// TIA Portal project "PROCESS OUTPUT" (V19)

(* hardware
DEVICE "SIMATIC 1200 station_1"  S71200.Device
   slot 0: "S7-1200 rack"  Rack  V1.0
   slot 1: "PLC_1"  CPU 1214C DC/DC/DC  6ES7 214-1AG40-0XB0  V4.0
   slot 3: "AQ1 x 12 bits_1"  6ES7 232-4HA30-0XB0  V1.0
DEVICE "HMI_1"  KTP600 Basic color PN
   slot 0: "HMI"  HMI  6AV6 647-0AD11-3AX0  12.0.0.0
   slot 1: "HMI_RT_1"  KTP600 Basic color PN  6AV6 647-0AD11-3AX0  12.0.0.0
   slot 5: "IE_CP_1"  PROFINET Interface  IE_CP  V7.1.0
      slot 1: "PROFINET_Interface_1"  PROFINET Interface
         slot 1: "PORT_1"  Port  1.0.0.0
*)

// ===== PLC "PLC_1"  CPU 1214C DC/DC/DC =====

VAR_GLOBAL   // PLC tag table "Default tag table"
   "SW_START" AT %I0.0 : Bool;   // START Momentary N. O. Pushbutton
   "PROCESS_OUT" AT %Q0.0 : Bool;   // Process Output
END_VAR

DATA_BLOCK "Data_block_Process"   // DB1
{ S7_Optimized_Access := 'TRUE' }
VERSION : 0.1
   VAR
      A_MATERIAL_MULTIPLIER : Real;   // Material A Multiplier
      B_MATERIAL_MULTIPLIER : Real;   // Material B Multiplier
      C_MATERIAL_MULTIPLIER : Real;   // Material C Multiplier
      D_MATERIAL_MULTIPLIER : Real;   // Material D Multiplier
      MATERIAL_MULTI_VALUE : Real;   // Material Multiplier Value
      PROCESS_VALUE : Real;   // Process Value
   END_VAR
BEGIN
END_DATA_BLOCK

DATA_BLOCK "Data_block_HMI"   // DB3
{ S7_Optimized_Access := 'TRUE' }
VERSION : 0.1
   VAR
      HMI_TYPE_SHEEt : Int;   // Operator Panel Pushbuttons Value for Sheet Type
      HMI_NUM_SHEET : Int;   // Operator Panel Pushbuttons Value for Number of Sheets
      HMI_PT_PROCESS_TIME : Real;   // Operator Panel Process Preset Time Value for program Timer Preset.
      HMI_ET_PROCESS_TIME : Real;   // Operator Panel Process Elapsed Time Value for Program Timer Elapsed.
      HMI_SW_START : Bool;   // HMI Start Switch
   END_VAR
BEGIN
END_DATA_BLOCK

// folder: System blocks/Program resources

DATA_BLOCK "PROCESS_TIMER"   // DB2
{ S7_Optimized_Access := 'TRUE' }
AUTHOR : Simatic
FAMILY : IEC
NAME : IEC_TMR
VERSION : 1.0
// stored: InstanceOfName IEC_TIMER
"IEC_TIMER"
BEGIN
END_DATA_BLOCK

// folder: (top level)

FUNCTION "Block_Time_Convert" : Void   // FC1, LAD
{ S7_Optimized_Access := 'TRUE' }
VERSION : 0.1
BEGIN
END_FUNCTION

FUNCTION "Block_HMI" : Void   // FC2, LAD
{ S7_Optimized_Access := 'TRUE' }
VERSION : 0.1
BEGIN
END_FUNCTION

FUNCTION "Block Time_Convert" : Void   // FC3, FBD
{ S7_Optimized_Access := 'TRUE' }
VERSION : 0.1
   VAR_INPUT
      IEC_TIMER_PT : Time;   // Timer PT Converted to Integer
      IEC_TIMER_ET : Time;   // Timer PT Converted to Real
   END_VAR
   VAR_OUTPUT
      IEC_TIMER_REAL_PT : Real;   // Timer ET Converted to Integer
      IEC_TIMER_REAL_ET : Real;   // Timer ET Converted to Real
   END_VAR
   VAR_TEMP
      PT_DINT : DInt;   // Preset Value as Integer
      PT_REAL : Real;   // Preset Value as Real
      ET_DINT : DInt;   // Elapsed Value as Integer
      ET_REAL : Real;   // Elapsed Value as Real
   END_VAR
BEGIN
END_FUNCTION

ORGANIZATION_BLOCK "Main"   // OB1, LAD, ProgramCycle
TITLE = "Main Program Sweep (Cycle)"
{ S7_Optimized_Access := 'TRUE' }
VERSION : 0.1
BEGIN
END_ORGANIZATION_BLOCK

(* ===== HMI "HMI_RT_1" =====
system functions are stored by id; their names below are inferred from use
connection "HMI_connection": ETHERNET, SMART_S7_1200_OMS

HMI tags "Default tag table"
   "Data_block_Process_A_MATERIAL_MULTIPLIER" : Real = PLC Data_block_Process.A_MATERIAL_MULTIPLIER, 1 s
   "Data_block_Process_B_MATERIAL_MULTIPLIER" : Real = PLC Data_block_Process.B_MATERIAL_MULTIPLIER, 1 s
   "Data_block_Process_C_MATERIAL_MULTIPLIER" : Real = PLC Data_block_Process.C_MATERIAL_MULTIPLIER, 1 s
   "Data_block_Process_D_MATERIAL_MULTIPLIER" : Real = PLC Data_block_Process.D_MATERIAL_MULTIPLIER, 1 s
   "Data_block_HMI_HMI_SW_START" : Bool = PLC Data_block_HMI.HMI_SW_START, 1 s
   "PROCESS_OUT" : Bool = PLC PROCESS_OUT AT %Q0.0, 1 s
   "Data_block_HMI_HMI_PT_PROCESS_TIME" : Real = PLC Data_block_HMI.HMI_PT_PROCESS_TIME, 1 s
   "Data_block_HMI_HMI_ET_PROCESS_TIME" : Real = PLC Data_block_HMI.HMI_ET_PROCESS_TIME, 1 s
   "Data_block_HMI_HMI_TYPE_SHEET" : Int = PLC Data_block_HMI.HMI_TYPE_SHEEt, 1 s
   "Data_block_HMI_HMI_NUM_SHEET" : Int = PLC Data_block_HMI.HMI_NUM_SHEET, 1 s

Template "Template_1" 320x240
   Button "Template_" at 267,201 size 51x37; TextOff 'ExitRuntime'; PictureOff "ExitRuntime_HMI_1"; PictureOn "ExitRuntime_HMI_1"
      on Release: StopRuntime(0)

screen "Root screen" 320x240, template "Template_1"
   Softkey "Softkey_F6" at 266,202 size 53x38
      on KeyDown: StopRuntime(0)
   GraphicIOField "PlotLight_Round_G" at 253,21 size 50x50; PictureOn "PilotLight_Round_G_On_256c"; PictureOff "PilotLight_Round_R_On_256c"
      ProcessValue <- "PROCESS_OUT"
   IOField "I/O field_1" at 194,108 size 74x26; FormatPattern 99.99
      ProcessValue <- "Data_block_HMI_HMI_PT_PROCESS_TIME"
   Button "Button_1" at 166,38 size 82x32; TextOff 'START'
      on Press: SetBit("Data_block_HMI_HMI_SW_START")
      on Release: ResetBit("Data_block_HMI_HMI_SW_START")
   IOField "I/O field_2" at 194,158 size 74x26; FormatPattern 99.99
      ProcessValue <- "Data_block_HMI_HMI_ET_PROCESS_TIME"
   TextField "Text field_1" at 23,8 size 33x18; Text 'TYPE'
   TextField "Text field_2" at 86,8 size 53x18; Text 'NUMBER'
   TextField "Text field_3" at 178,17 size 59x18; Text 'PROCESS'
   TextField "Text field_4" at 205,88 size 48x18; Text 'PRESET'
   TextField "Text field_5" at 170,138 size 118x18; Text 'CURRENT ELASPED'
   Switch "Switch_1" at 94,31 size 34x34; CaptionText 'Switch'; TextOff '2'; TextOn '2'
      ProcessValue <- "Data_block_HMI_HMI_NUM_SHEET"
   Switch "Switch_2" at 94,71 size 34x34; CaptionText 'Switch'; TextOff '3'; TextOn '3'
      ProcessValue <- "Data_block_HMI_HMI_NUM_SHEET"
   Switch "Switch_4" at 94,111 size 34x34; CaptionText 'Switch'; TextOff '4'; TextOn '4'
      ProcessValue <- "Data_block_HMI_HMI_NUM_SHEET"
   Switch "Switch_5" at 94,151 size 34x34; CaptionText 'Switch'; TextOff '5'; TextOn '5'
      ProcessValue <- "Data_block_HMI_HMI_NUM_SHEET"
   Switch "Switch_6" at 94,191 size 34x34; CaptionText 'Switch'; TextOff '6'; TextOn '6'
      ProcessValue <- "Data_block_HMI_HMI_NUM_SHEET"
   Switch "Switch_3" at 21,31 size 34x34; CaptionText 'Switch'; TextOff 'A'; TextOn 'A'
      ProcessValue <- "Data_block_HMI_HMI_TYPE_SHEET"
   Switch "Switch_7" at 21,71 size 34x34; CaptionText 'Switch'; TextOff 'B'; TextOn 'B'
      ProcessValue <- "Data_block_HMI_HMI_TYPE_SHEET"
   Switch "Switch_8" at 21,111 size 34x34; CaptionText 'Switch'; TextOff 'C'; TextOn 'C'
      ProcessValue <- "Data_block_HMI_HMI_TYPE_SHEET"
   Switch "Switch_9" at 21,151 size 34x34; CaptionText 'Switch'; TextOff 'D'; TextOn 'D'
      ProcessValue <- "Data_block_HMI_HMI_TYPE_SHEET"
   Button "Button_2" at 1,201 size 51x37; TextOff 'PANEL 2'
      on Release: ActivateScreen("Screen_2", 0)
   Softkey "Softkey_F1" at 1,202 size 53x38
      on KeyDown: ActivateScreen("Screen_2", 0)

screen "Screen_2" 320x240
   IOField "I/O field_1" at 162,41 size 105x28; FormatPattern 99.99
      ProcessValue <- "Data_block_Process_A_MATERIAL_MULTIPLIER"
   IOField "I/O field_2" at 162,82 size 105x28; FormatPattern 99.99
      ProcessValue <- "Data_block_Process_B_MATERIAL_MULTIPLIER"
   IOField "I/O field_3" at 162,123 size 105x28; FormatPattern 99.99
      ProcessValue <- "Data_block_Process_C_MATERIAL_MULTIPLIER"
   IOField "I/O field_4" at 162,164 size 105x28; FormatPattern 99.99
      ProcessValue <- "Data_block_Process_D_MATERIAL_MULTIPLIER"
   Button "Button_1" at 1,201 size 51x37; TextOff 'MAIN'
      on Release: ActivateScreen("Root screen", 0)
   TextField "Text field_1" at 56,8 size 209x20; Text 'MULTIPLIER VALUE SET-UP'
   TextField "Text field_2" at 59,45 size 94x20; Text 'MATERIAL A'
   TextField "Text field_3" at 59,86 size 94x20; Text 'MATERIAL B'
   TextField "Text field_4" at 59,127 size 94x20; Text 'MATERIAL C'
   TextField "Text field_5" at 59,168 size 95x20; Text 'MATERIAL D'
   Softkey "Softkey_F1" at 1,202 size 53x38
      on KeyDown: ActivateScreen("Root screen", 0)
*)